PROGRAM Proces_1
VAR

Step		: UINT;	

// INputs
Start			: BOOL;
Beker_aanwezig	: BOOL;
Bonen_aanwezig	: BOOL;
Melk_aanwezig	: BOOL;
Voldoende_water	: BOOL;
Start_Spoelen :BOOL;	


// Outputs
Led_ready_start		: BOOL;
Melk_verwarming		: BOOL;
Melk_pomp			: BOOL;
Bonen_malen			: BOOL;
Water_pomp			: BOOL;
Spoelen		: BOOL; 









// Timers
Timer 		: TON;
Timer2 		: TON;
Timer3 		: TON;
Timer4 		: TON;
END_VAR



// Statemachine
CASE Step OF
	0: //Init stap 0
		IF GVL.Power_ON = TRUE THEN
			Step				:=10;
		END_IF
	

	10: // Spoelen machine 
	Timer(IN:=TRUE, PT:=T#5S);
	Start_Spoelen := TRUE;
	Spoelen := functie(Spoelen_start := Start_Spoelen, Timer);	

	
	IF Spoelen = TRUE THEN
		Step		:=20;
	END_IF

	20: // klaar om te starten
	Timer(IN:=FALSE, PT:=T#5S);
	//spoelen := FALSE;
	IF Bonen_aanwezig = TRUE  AND Melk_aanwezig = TRUE AND Voldoende_water THEN
		Led_ready_start := TRUE;
		Step 	:= 30;
	END_IF
	
	
	30: // Wanneer beker aanwezig is en op strat word geklikt. Melk word verwarmt en bonen worden gemalen.
	IF Start = TRUE AND Beker_aanwezig = TRUE THEN
		Led_ready_start := FALSE;
		Melk_verwarming	:= TRUE;
		Bonen_malen		:= TRUE;
		Timer2(IN:=TRUE, PT:=T#5S);	
	END_IF
	
	
	IF Timer2.Q = TRUE THEN
		Timer2(IN:=FALSE);
		Start := FALSE;
		Step	:= 40;
	END_IF
	

	40: // na 5 sec gaat bonen malen uit en de melk pomp aan voor toevoegen melk.
	Bonen_malen		:= FALSE;
	Melk_pomp		:= TRUE;
	
	Timer3(IN:=TRUE, PT:=T#5S);
	
	IF Timer3.Q = TRUE THEN
		Timer3(IN:=FALSE);
		Step	:= 50;
	END_IF	
	
	50: // na 5 sec melk verwarming en pomp gaan uit. water word door de bonen gepompt.
	Melk_verwarming	:= FALSE;
	Melk_pomp		:= FALSE;
	Water_pomp		:= TRUE;
	
	Timer4(IN:=TRUE, PT:=T#5S);
	
	IF Timer4.Q = TRUE THEN
		Timer4(IN:=FALSE);
		Step	:= 60;
	END_IF

	60: 
	Water_pomp		:= FALSE;
	
	IF Beker_aanwezig = FALSE THEN
		Step	:= 10;
	END_IF
END_CASE

END_PROGRAM

(* stored: Version 1.1.0.1, ProductVersion 3.1.4024.12
   POU Proces_1: Id {ecdb4a31-0add-4a42-99fb-f6ca525697d9}, SpecialFunc None *)
